(* IEC 61131-3 sources: teller/JD_Teller_LC2_V11/Class/Free_Jamdetector, 1 file *)

(* ---- Free_Jamdetector.st ---- *)
(*!
<Class
	Name               = "Free_Jamdetector"
	Revision           = "1.1"
	RealtimeTask       = "true"
	DefRealtime        = "1 ms"
	CyclicTask         = "true"
	DefCyclictime      = "50 ms"
	BackgroundTask     = "false"
	Sigmatek           = "false"
	OSInterface        = "false"
	HighPriority       = "false"
	Automatic          = "false"
	UpdateMode         = "Prescan"
	SharedCommandTable = "true"
	Objectsize         = "(570,900)">
	<Channels>
		<Server Name="iEncDiv" Visualized="true" Initialize="false" WriteProtected="false" Retentive="false" Comment="SS"/>
		<Server Name="iEncMulti" Visualized="true" Initialize="false" WriteProtected="false" Retentive="false" Comment="SS"/>
		<Server Name="iJamBoxlength" Visualized="true" Initialize="false" WriteProtected="false" Retentive="false"/>
		<Server Name="iJamBoxlength_Max" Visualized="true" Initialize="false" WriteProtected="false" Retentive="false"/>
		<Server Name="iJamBoxlength_Min" Visualized="true" Initialize="false" WriteProtected="false" Retentive="false"/>
		<Server Name="iJamReset" Visualized="false" Initialize="false" WriteProtected="false" Retentive="false"/>
		<Server Name="iMinSpot" Visualized="true" Initialize="false" WriteProtected="false" Retentive="false" Comment="SS&#13;&#10;"/>
		<Server Name="iSExtraBox" Visualized="true" Initialize="false" WriteProtected="false" Retentive="false"/>
		<Server Name="oJamDet" Visualized="false" Initialize="false" WriteProtected="true" Retentive="false"/>
		<Server Name="oSensorHW" Visualized="true" Initialize="false" WriteProtected="true" Retentive="false" Comment="OS"/>
		<Server Name="oSpeed" Visualized="true" Initialize="false" WriteProtected="true" Retentive="false" Comment="OS"/>
		<Server Name="Server0" Visualized="true" Initialize="false" WriteProtected="true" Retentive="false"/>
		<Server Name="TaskOnOff" Visualized="false" Initialize="false" WriteProtected="false" Retentive="false"/>
		<Server Name="vSection" Visualized="true" Initialize="false" WriteProtected="false" Retentive="false"/>
		<Server Name="vUnit" Visualized="true" Initialize="false" WriteProtected="false" Retentive="false"/>
		<Client Name="iEncoder" Required="false" Internal="false"/>
		<Client Name="iSensor" Required="false" Internal="false"/>
		<Client Name="rEncdiv" Required="true" Internal="true"/>
		<Client Name="rEncmulti" Required="true" Internal="true"/>
		<Client Name="rJamBoxlength" Required="true" Internal="true"/>
		<Client Name="rMinSpot" Required="true" Internal="true"/>
		<Client Name="rSExtraBox" Required="true" Internal="true"/>
		<Client Name="rvSection" Required="true" Internal="true"/>
		<Client Name="rvUnit" Required="true" Internal="true"/>
	</Channels>
	<RevDoku>
		<Owner Company="JD" Author="JVD"/>
		<Dokumentation Revision="1.1" Date="2013-09-21" Author="JVD" Company="JD" Description="Return state opgelost"/>
		<Dokumentation Revision="1.0" Date="2012-07-04" Author="JVD" Company="JD" Description="Taskmanager included"/>
	</RevDoku>
	<Network Name="Free_Jamdetector">
		<!-- List of Components in this network -->
		<Components>
			<Object
				Name       = "rEncdiv"
				Class      = "Ram"
				Position   = "(270,450)"
				Visualized = "true">
				<Channels>
					<Server Name="Data"/>
				</Channels>
			</Object>
			<Object
				Name       = "rEncmulti"
				Class      = "Ram"
				Position   = "(270,300)"
				Visualized = "true">
				<Channels>
					<Server Name="Data"/>
				</Channels>
			</Object>
			<Object
				Name       = "rJamBoxlength"
				Class      = "Ram"
				Position   = "(270,750)"
				Visualized = "true">
				<Channels>
					<Server Name="Data"/>
				</Channels>
			</Object>
			<Object
				Name       = "rMinSpot"
				Class      = "Ram"
				Position   = "(270,150)"
				Visualized = "true">
				<Channels>
					<Server Name="Data"/>
				</Channels>
			</Object>
			<Object
				Name       = "rSExtraBox"
				Class      = "Ram"
				Position   = "(270,600)"
				Visualized = "true">
				<Channels>
					<Server Name="Data"/>
				</Channels>
			</Object>
			<Object
				Name       = "rvSection"
				Class      = "Ram"
				Position   = "(270,900)"
				Visualized = "true">
				<Channels>
					<Server Name="Data"/>
				</Channels>
			</Object>
			<Object
				Name       = "rvUnit"
				Class      = "Ram"
				Position   = "(270,1050)"
				Visualized = "true">
				<Channels>
					<Server Name="Data"/>
				</Channels>
			</Object>
		</Components>
		<Comments>
		</Comments>
		<!-- List of Connections in this network -->
		<Connections>
			<Connection Source="this.rEncmulti" Destination="rEncmulti.Data"/>
			<Connection Source="this.rEncdiv" Destination="rEncdiv.Data"/>
			<Connection Source="this.rJamBoxlength" Destination="rJamBoxlength.Data"/>
			<Connection Source="this.rvSection" Destination="rvSection.Data"/>
			<Connection Source="this.rvUnit" Destination="rvUnit.Data"/>
			<Connection Source="this.rMinSpot" Destination="rMinSpot.Data"/>
			<Connection Source="this.rSExtraBox" Destination="rSExtraBox.Data"/>
		</Connections>
		<!-- Headerfiles -->
		<Options>
		</Options>
	</Network>
</Class>
*)
Free_Jamdetector : CLASS
  //Servers:
	Server0 	: SvrChCmd_DINT;
	TaskOnOff 	: SvrCh_DINT;
	iMinSpot 	: SvrCh_DINT;
	oSensorHW 	: SvrCh_DINT;
	oSpeed 	: SvrCh_DINT;
	iEncMulti 	: SvrCh_DINT;
	iEncDiv 	: SvrCh_DINT;
	iSExtraBox 	: SvrCh_DINT;
	oJamDet 	: SvrCh_DINT;
	iJamReset 	: SvrCh_DINT;
	iJamBoxlength 	: SvrCh_DINT;
	vSection 	: SvrCh_DINT;
	vUnit 	: SvrCh_DINT;
	iJamBoxlength_Min 	: SvrCh_DINT;
	iJamBoxlength_Max 	: SvrCh_DINT;
  //Clients:
	rEncmulti 	: CltChCmd_Ram;
	rEncdiv 	: CltChCmd_Ram;
	rMinSpot 	: CltChCmd_Ram;
	iEncoder 	: CltCh_DINT;
	iSensor 	: CltCh_DINT;
	rSExtraBox 	: CltChCmd_Ram;
	rJamBoxlength 	: CltChCmd_Ram;
	rvSection 	: CltChCmd_Ram;
	rvUnit 	: CltChCmd_Ram;
  //Variables:
		Enc 	: Encoder1;
		sensor 	: tSensor;
		Jam 	: tJam;
		OSpeedie 	: tOspeed;
  //Functions:

	FUNCTION VIRTUAL GLOBAL Init;

	FUNCTION VIRTUAL GLOBAL CyWork
		VAR_INPUT
			EAX 	: UDINT;
		END_VAR
		VAR_OUTPUT
			state (EAX) 	: UDINT;
		END_VAR;

	FUNCTION VIRTUAL GLOBAL RtWork
		VAR_INPUT
			EAX 	: UDINT := EAX;
		END_VAR
		VAR_OUTPUT
			state (EAX) 	: UDINT;
		END_VAR;
  //Tables:
	FUNCTION @STD
		VAR_OUTPUT
			ret_code	: CONFSTATES;
		END_VAR;
	FUNCTION GLOBAL TAB @CT_;
END_CLASS;

#pragma using Ram

//************************************************************************

FUNCTION VIRTUAL GLOBAL Free_Jamdetector::Init

	if _firstscan then

//    //geheugen uitlezen
      rEncmulti := rEncmulti.Read();
      rEncdiv := rEncdiv.Read();
      rMinSpot := rMinSpot.Read();
      rSExtraBox := rSExtraBox.Read();
      rJamBoxlength := rJamBoxlength.Read();
      rvSection := rvSection.Read();
      rvUnit := rvUnit.Read();

      iEncMulti.Write(rEncmulti);
      iEncDiv.Write(rEncdiv);
      iMinSpot.Write(rMinSpot);
      iSExtraBox.Write(rSExtraBox);
      iJamBoxlength.Write(rJamBoxlength);
      vSection.Write(rvSection);
      vUnit.Write(rvUnit);
      iJamBoxlength_Max:=2000;
      iJamBoxlength_Min:=0;

	end_if;

END_FUNCTION

FUNCTION VIRTUAL GLOBAL Free_Jamdetector::RtWork
	VAR_INPUT
		EAX 	: UDINT;
	END_VAR
	VAR_OUTPUT
		state (EAX) 	: UDINT;
	END_VAR

//Als in de machine setup de functie is geselelecteerd wordt de code uitgevoerd
  if  TaskOnOff then

//inlezen van de sensors

            iSensor := iSensor.Read();
            oSensorHW :=iSensor;
            oSensorHW.Write(iSensor);

//Divider mag niet 0 zijn!
        if iEncDiv = 0 then
           iEncDiv:=1;
        end_if;

//inlezen van de encoder

          iEncoder:=iEncoder.Read();

          Enc.EncoderDelta := iEncoder - Enc.EncoderOld;
          Enc.EncoderOld := iEncoder;

          Enc.Multi := iEncMulti;
          Enc.Divider := iEncDiv;

          Enc.SpeedDelta := ((Enc.EncoderDelta * encres * enc.Multi) / enc.Divider);

//one shot op de ingang

          case Sensor.MinimaalSSW of

          0:
            if  iSensor = 1 then
                Sensor.MinimaleCounter:=0;
                Sensor.Din:=0;
                Sensor.MinimaalSSW+=1;
            end_if;

          1:

            Sensor.MinimaleCounter+= Enc.SpeedDelta;

            if  Sensor.MinimaleCounter > (iMinSpot * encres) then
                if  iSensor = 1 then
                    Sensor.Din:=1;
                    Sensor.MinimaalSSW+=1;
                else
                    Sensor.MinimaalSSW:=0;
                end_if;

            end_if;

          2:
                Sensor.Din:=0;
            if  iSensor = 0 then
                Sensor.MinimaalSSW:=0;
            end_if;

          end_case;

//Jam

             if iJamBoxlength <> 0 then

                  case Jam.CaseJam of

                  0: //controleren of aan de snipper beveiliging is voldaan
                     if Sensor.Din then
                        Jam.CaseJam += 1;
                        Jam.JamPos :=  iMinSpot * encres;
                     end_if;

                  1: //Controle op Jamdetect
                     //Kijken of de sensor hoog is na de ingestelde Boxlengte en extra waarde

                        Jam.JamPos += Enc.SpeedDelta;
                        Jam.JamBoxlength := (iJamBoxlength + iSExtraBox) * encres;

                         if   Jam.JamPos > Jam.JamBoxlength then //De Jampos loopt nu mee
                            if   iSensor then
                                Jam.JamDetection := 1;
                                oJamdet := jam.Jamdetection;
                                oJamdet.Write(oJamdet);
                                Jam.CaseJam += 1;
                            else                                //Geen Jamdetect!!
                                Jam.JamDetection := 0;   //Geen Jamdetect, terug naar stap 0 en wachten op een nieuwe doos
                                oJamdet := jam.Jamdetection;
                                oJamdet.Write(oJamdet);
                                Jam.CaseJam := 0;
                            end_if;

                         end_if;

                  2:  //Jam, reset is nodig om verder te gaan.
                     oJamdet.Write(jam.Jamdetection);

                     if iJamReset then
                        Jam.JamDetection := 0;
                        oJamdet := jam.Jamdetection;
                        oJamdet.Write(oJamdet);
                        Jam.CaseJam:=0;
                        Jam.Jampos:=0;
                     end_if;

                   end_case;
              end_if;

  end_if;

  state := READY;
END_FUNCTION //VIRTUAL GLOBAL Infeed::RtWork

FUNCTION VIRTUAL GLOBAL Free_Jamdetector::CyWork
	VAR_INPUT
		EAX 	: UDINT;
	END_VAR
	VAR_OUTPUT
		state (EAX) 	: UDINT;
	END_VAR

//Als in de machine setup de functie is geselelecteerd wordt de code uitgevoerd
  if  TaskOnOff then
   //Servers in Ram opslaan

      iEncMulti := iEncMulti.Read();
      rEncmulti.Write(iEncMulti);
      iEncDiv:=iEncDiv.Read();
      rEncdiv.Write(iEncDiv);
      iMinSpot := iMinSpot.Read();
      rMinSpot.Write(iMinSpot);
      iSExtraBox := iSExtraBox.Read();
      rSExtraBox.Write(iSExtraBox);
      iJamBoxlength := iJamBoxlength.Read();
      rJamBoxlength.Write(iJamBoxlength);
      vSection := vSection.Read();
      rvSection.Write(vSection);
      vUnit := vUnit.Read();
      rvUnit.Write(vUnit);

          OSpeedie.EncIn :=iEncoder.Read();
          ospeedie.EncDelta := OSpeedie.EncIn - OSpeedie.EncOud;
          OSpeedie.EncOud := OSpeedie.EncIn;
          oSpeed := to_dint((to_Real(ospeedie.EncDelta) * 60 * To_Real(iEncMulti)) / (to_Real(iEncDiv)*50));

      //oSpeed := ((enc.SpeedDelta  * 60) / encres);   //mm/ms  vermenigvuldigen met 60000 / 1000

  end_if;

	state := READY;

END_FUNCTION
